// SIMATIC STEP 7 (V5.x) project Estacionamiento
// CPU: CPU 315-2 DP
// CPU: CPU 315-2 DP
// station: Hardware
// station: Estación 1
// station: P_ADR_BUS
// station: Hardware
// station: Estación 2
// station: P_ADR_BUS
// program: 2P
// program: Programa S7(6)
// program: Programa S7(7)

// (several symbol tables fit these blocks; global names not applied)

// FC 1: know-how protected block, not included

// FC 2: know-how protected block, not included

ORGANIZATION_BLOCK OB 1
TITLE = "Main Program Sweep (Cycle)"
VERSION : 0.1
VAR_TEMP
  OB1_EV_CLASS : BYTE ;	//Bits 0-3 = 1 (Coming event), Bits 4-7 = 1 (Event class 1)
  OB1_SCAN_1 : BYTE ;	//1 (Cold restart scan 1 of OB 1), 3 (Scan 2-n of OB 1)
  OB1_PRIORITY : BYTE ;	//Priority of OB Execution
  OB1_OB_NUMBR : BYTE ;	//1 (Organization block 1, OB1)
  OB1_RESERVED_1 : BYTE ;	//Reserved for system
  OB1_RESERVED_2 : BYTE ;	//Reserved for system
  OB1_PREV_CYCLE : INT ;	//Cycle time of previous OB1 scan (milliseconds)
  OB1_MIN_CYCLE : INT ;	//Minimum cycle time of OB1 (milliseconds)
  OB1_MAX_CYCLE : INT ;	//Maximum cycle time of OB1 (milliseconds)
  OB1_DATE_TIME : DATE_AND_TIME ;	//Date and time OB1 started
END_VAR
BEGIN
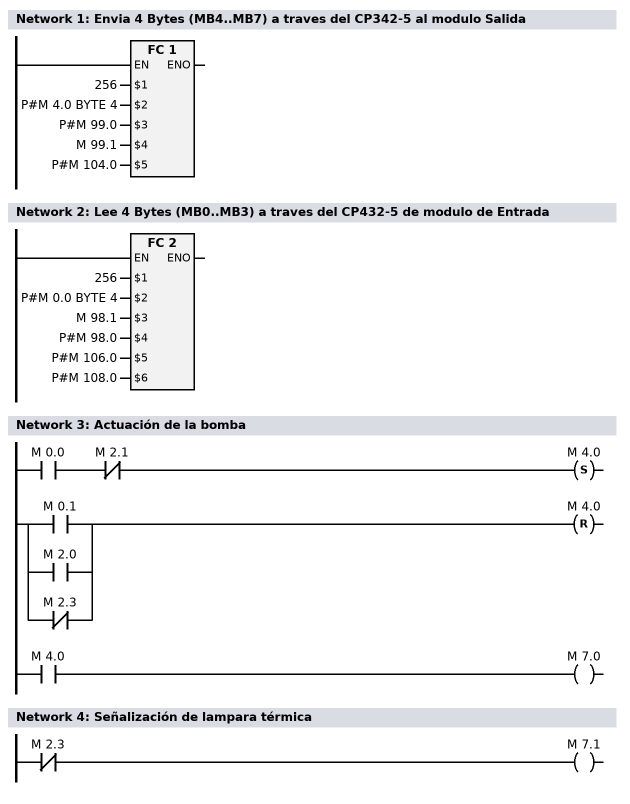
NETWORK
TITLE = Envia 4 Bytes (MB4..MB7) a traves del CP342-5 al modulo Salida
      CALL  FC 1 (
           $1                       := 256,
           $2                       := P#M 4.0 BYTE 4,
           $3                       := P#M 99.0,
           $4                       := M 99.1,
           $5                       := P#M 104.0);
      NOP   0;
NETWORK
TITLE = Lee 4 Bytes (MB0..MB3) a traves del CP432-5 de modulo de Entrada
      CALL  FC 2 (
           $1                       := 256,
           $2                       := P#M 0.0 BYTE 4,
           $3                       := M 98.1,
           $4                       := P#M 98.0,
           $5                       := P#M 106.0,
           $6                       := P#M 108.0);
      NOP   0;
NETWORK
TITLE = Actuación de la bomba
//Importante: Considerando el pulsador start tiene 
//autoretención. 
//Se inicia el sistema presionando el boton de start, 
//si el sensor bajo no detecta agua la bomba debe activarse.
//Si el sensor de alto detecta agua se debe apagar la bomba.
//Si se presiona el boton STOP la bomba debe parar.
//Si el sensor térmico esta activo tambien debe parar
//la bomba 
      A     M 0.0;
      AN    M 2.1;
      S     M 4.0;
      A(;
      O     M 0.1;
      O     M 2.0;
      ON    M 2.3;
      );
      R     M 4.0;
      A     M 4.0;
      =     M 7.0;
NETWORK
TITLE = Señalización de lampara térmica
//Si el sensor térmico esta activo se enciende la 
//señalización del Térmico
      AN    M 2.3;
      =     M 7.1;
NETWORK
TITLE =
END_ORGANIZATION_BLOCK

SYMBOL_TABLE
"Cuenta"	C 0	COUNTER	// Cantidad de vehículos estacionados
"DP_SEND"	FC 1	FC 1	// DP-SEND-Function for  SIMATIC NET CPs
"DP_RECV"	FC 2	FC 2	// DP-RECV-Function for  SIMATIC NET CPs
"ON/OFF Fisico"	I 0.0	BOOL	// Switch para modificar estado de la marca ON/OFF
"Reset Fisico"	I 0.1	BOOL	// Botón para resetear el contador
"Cont Entrada"	M 0.0	BOOL	// Aumenta el contador en uno al activarse (Corresponde con el I0.0)
"Cont Salida"	M 0.1	BOOL	// Disminuye el contador en uno al activarse (Corresponde con el I0.1)
"Lámpara Libre"	M 4.1	BOOL	// Se activa mientras estén menos de 20 vehículos dentro del estacionamiento (Q0.1)
"Lámpara Ocupado"	M 4.2	BOOL	// Se activa mientras estén 20 vehículos dentro del estacionamiento (Q0.2)
"Abrir"	M 5.0	BOOL	// Botón que libera el paso (Q1.0, en lugar del Q0.0 planteado inicialmente)
"Cerrar"	M 5.1	BOOL	// Botón que cierra el paso (Q1.1, en lugar del Q0.0 planteado inicialmente)
"ON/OFF"	M 30.0	BOOL	// Se activa el Sistema (ON) o cierra la barrera y conserva la cuenta (OFF) (input)
"Reset"	M 30.1	BOOL	// Vuelve a cero el contador (input físico o lógico)
"Marca Pizcando"	M 32.0	BOOL	// Para el pizcando de la luz
"Contador"	MW 102	WORD	// Cantidad de vehículos estacionados
"Cycle Execution"	OB 1	OB 1
"Hora"	QW 0	WORD
"Minuto"	QW 2	WORD
"READ_CLK"	SFC 1	SFC 1	// Read System Clock
"Temp"	T 0	TIMER	// Para la luz intermitente
"Temp1"	T 1	TIMER	// Para luz intermitente 2
END_SYMBOL_TABLE

// FC 1: know-how protected block, not included

// FC 2: know-how protected block, not included

ORGANIZATION_BLOCK "Cycle Execution"	// OB 1
TITLE = "Main Program Sweep (Cycle)"
VERSION : 0.1
VAR_TEMP
  OB1_EV_CLASS : BYTE ;	//Bits 0-3 = 1 (Coming event), Bits 4-7 = 1 (Event class 1)
  OB1_SCAN_1 : BYTE ;	//1 (Cold restart scan 1 of OB 1), 3 (Scan 2-n of OB 1)
  OB1_PRIORITY : BYTE ;	//Priority of OB Execution
  OB1_OB_NUMBR : BYTE ;	//1 (Organization block 1, OB1)
  OB1_RESERVED_1 : BYTE ;	//Reserved for system
  OB1_RESERVED_2 : BYTE ;	//Reserved for system
  OB1_PREV_CYCLE : INT ;	//Cycle time of previous OB1 scan (milliseconds)
  OB1_MIN_CYCLE : INT ;	//Minimum cycle time of OB1 (milliseconds)
  OB1_MAX_CYCLE : INT ;	//Maximum cycle time of OB1 (milliseconds)
  realtime : DATE_AND_TIME ;	//Date and time OB1 started
END_VAR
BEGIN
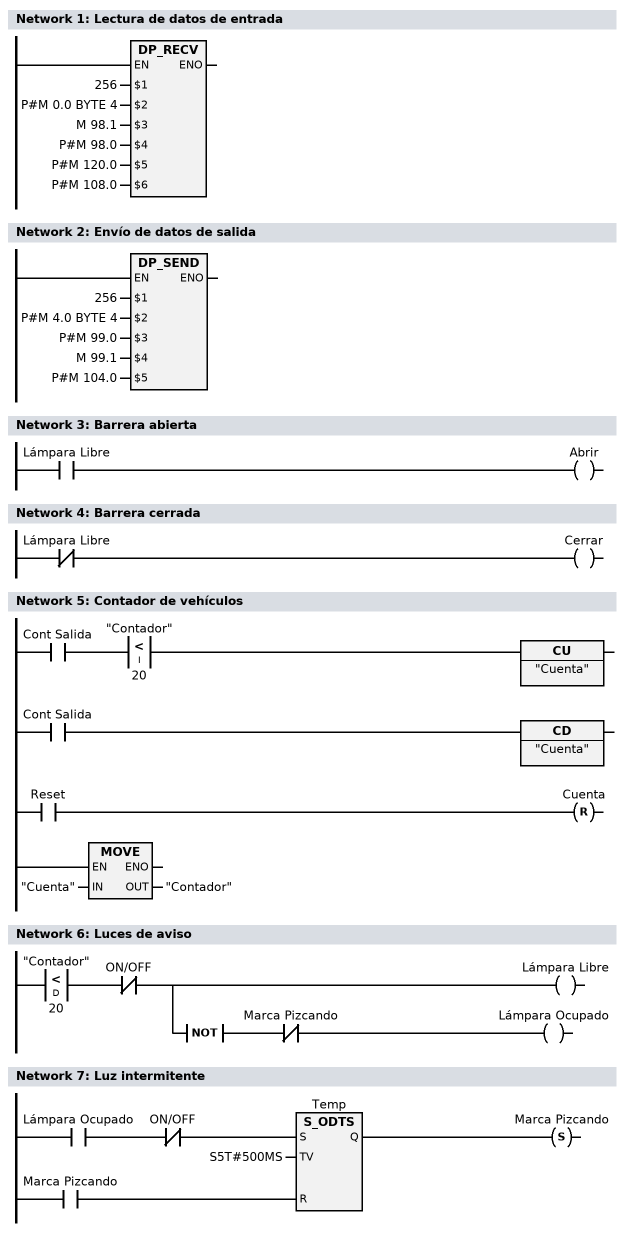
NETWORK
TITLE = Lectura de datos de entrada
      CALL  "DP_RECV" (
           $1                       := 256,
           $2                       := P#M 0.0 BYTE 4,
           $3                       := M 98.1,
           $4                       := P#M 98.0,
           $5                       := P#M 120.0,
           $6                       := P#M 108.0);
      NOP   0;
NETWORK
TITLE = Envío de datos de salida
      CALL  "DP_SEND" (
           $1                       := 256,
           $2                       := P#M 4.0 BYTE 4,
           $3                       := P#M 99.0,
           $4                       := M 99.1,
           $5                       := P#M 104.0);
      NOP   0;
NETWORK
TITLE = Barrera abierta
//Se mantine la barrera abierta mientras haya lugar ("lampara libre")
      A     "Lámpara Libre";
      =     "Abrir";
NETWORK
TITLE = Barrera cerrada
//Se mantine la barrera cerrada mientras no haya lugar ("lampara ocupada")
      AN    "Lámpara Libre";
      =     "Cerrar";
NETWORK
TITLE = Contador de vehículos
//Se realiza la deteccion de autos mediante los sensores del contador de 
//entrada/salida. El "cont entrada" aumente en 1 cuando ingresa un vehiculo;
//si el "Contador" es menor que la capacidad max. de autos (20)
//Y con el "cont salida" disminuye en 1 el "Contador" cuando sale un vehiculo.
      A     "Cont Salida";
      A(;
      L     "Contador";
      L     20;
      <I;
      );
      CU    "Cuenta";
      A     "Cont Salida";
      CD    "Cuenta";
      NOP   0;
      NOP   0;
      A     "Reset";
      R     "Cuenta";
      L     "Cuenta";
      T     "Contador";
      NOP   0;
      NOP   0;
NETWORK
TITLE = Luces de aviso
//Si el "Contador" es menor a 20 la "Lampara Libre" estara encendida
//y si llega a la capacidad maxima se enciende la "Lampara Ocupado" de 
//manera intermitente
      A(;
      L     "Contador";
      L     20;
      <D;
      );
      AN    "ON/OFF";
      =     L 20.0;
      A     L 20.0;
      BLD   102;
      =     "Lámpara Libre";
      A     L 20.0;
      NOT;
      AN    "Marca Pizcando";
      =     "Lámpara Ocupado";
NETWORK
TITLE = Luz intermitente
//Metodo por el cual se logra que la "Lampara Ocupado"
//se encienda de forma intermitente parte 1
      A     "Lámpara Ocupado";
      AN    "ON/OFF";
      L     S5T#500MS;
      SS    "Temp";
      A     "Marca Pizcando";
      R     "Temp";
      NOP   0;
      NOP   0;
      A     "Temp";
      S     "Marca Pizcando";
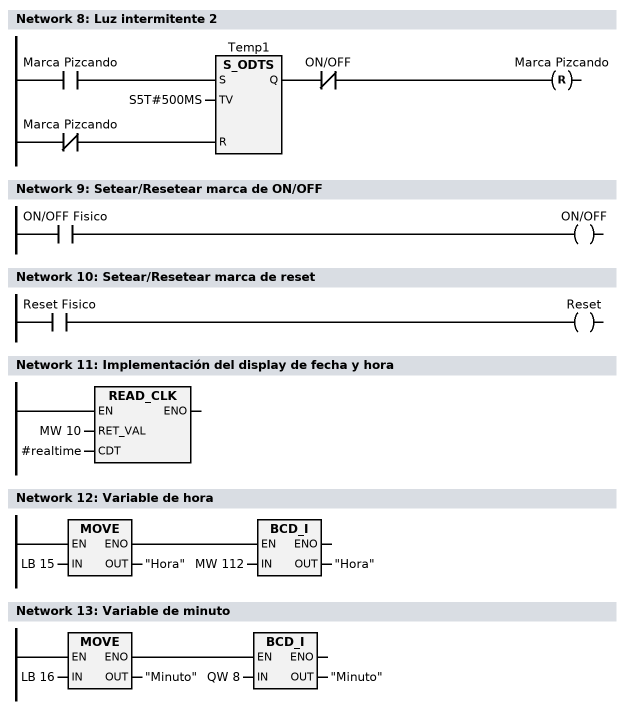
NETWORK
TITLE = Luz intermitente 2
//Metodo por el cual se logra que la "Lampara Ocupado"
//se encienda de forma intermitente parte 2
      A(;
      A     "Marca Pizcando";
      L     S5T#500MS;
      SS    "Temp1";
      AN    "Marca Pizcando";
      R     "Temp1";
      NOP   0;
      NOP   0;
      A     "Temp1";
      );
      AN    "ON/OFF";
      R     "Marca Pizcando";
NETWORK
TITLE = Setear/Resetear marca de ON/OFF
//Una vez que se cambia el valor del switch físico de on/off, una marca toma ese 
//valor. Este switch se encuentra del lado de la CPU.
      A     "ON/OFF Fisico";
      =     "ON/OFF";
NETWORK
TITLE = Setear/Resetear marca de reset
//Así como el switch de on/off, el botón físico de reset se encuentra del lado 
//del 
//operador (donde está el CPU), y la marca se activa mientras el botón esté 
//pulsado.
      A     "Reset Fisico";
      =     "Reset";
NETWORK
TITLE = Implementación del display de fecha y hora
//Los siguientes segmentos asignarán valores codificados en BCD del  
//hora y minuto para que estos sean mostrados del lado del 
//CPU, conectando estas salidas físicas a displays de 7 segmentos que reciban 
//números en BCD como entradas.
      CALL  "READ_CLK" (
           RET_VAL                  := MW 10,
           CDT                      := #realtime);
      NOP   0;
NETWORK
TITLE = Variable de hora
      A(;
      L     LB 15;
      T     "Hora";
      SET;
      SAVE;
      CLR;
      A     BR;
      );
      JNB   _001;
      L     MW 112;
      BTI;
      T     "Hora";
_001: NOP   0;
NETWORK
TITLE = Variable de minuto
      A(;
      L     LB 16;
      T     "Minuto";
      SET;
      SAVE;
      CLR;
      A     BR;
      );
      JNB   _002;
      L     QW 8;
      BTI;
      T     "Minuto";
_002: NOP   0;
END_ORGANIZATION_BLOCK

SYMBOL_TABLE
"DP_SEND"	FC 1	FC 1	// DP-SEND-Function for  SIMATIC NET CPs
"DP_RECV"	FC 2	FC 2	// DP-RECV-Function for  SIMATIC NET CPs
"AG_SEND"	FC 5	FC 5	// AG SEND
"AG_RECV"	FC 6	FC 6	// AG RECEIVE
"Cycle Execution"	OB 1	OB 1
"READ_CLK"	SFC 1	SFC 1	// Read System Clock
END_SYMBOL_TABLE

// FC 5: know-how protected block, not included

// FC 6: know-how protected block, not included

ORGANIZATION_BLOCK "Cycle Execution"	// OB 1
TITLE = "Main Program Sweep (Cycle)"
VERSION : 0.1
VAR_TEMP
  OB1_EV_CLASS : BYTE ;	//Bits 0-3 = 1 (Coming event), Bits 4-7 = 1 (Event class 1)
  OB1_SCAN_1 : BYTE ;	//1 (Cold restart scan 1 of OB 1), 3 (Scan 2-n of OB 1)
  OB1_PRIORITY : BYTE ;	//Priority of OB Execution
  OB1_OB_NUMBR : BYTE ;	//1 (Organization block 1, OB1)
  OB1_RESERVED_1 : BYTE ;	//Reserved for system
  OB1_RESERVED_2 : BYTE ;	//Reserved for system
  OB1_PREV_CYCLE : INT ;	//Cycle time of previous OB1 scan (milliseconds)
  OB1_MIN_CYCLE : INT ;	//Minimum cycle time of OB1 (milliseconds)
  OB1_MAX_CYCLE : INT ;	//Maximum cycle time of OB1 (milliseconds)
  realtime : DATE_AND_TIME ;	//Date and time OB1 started
END_VAR
BEGIN
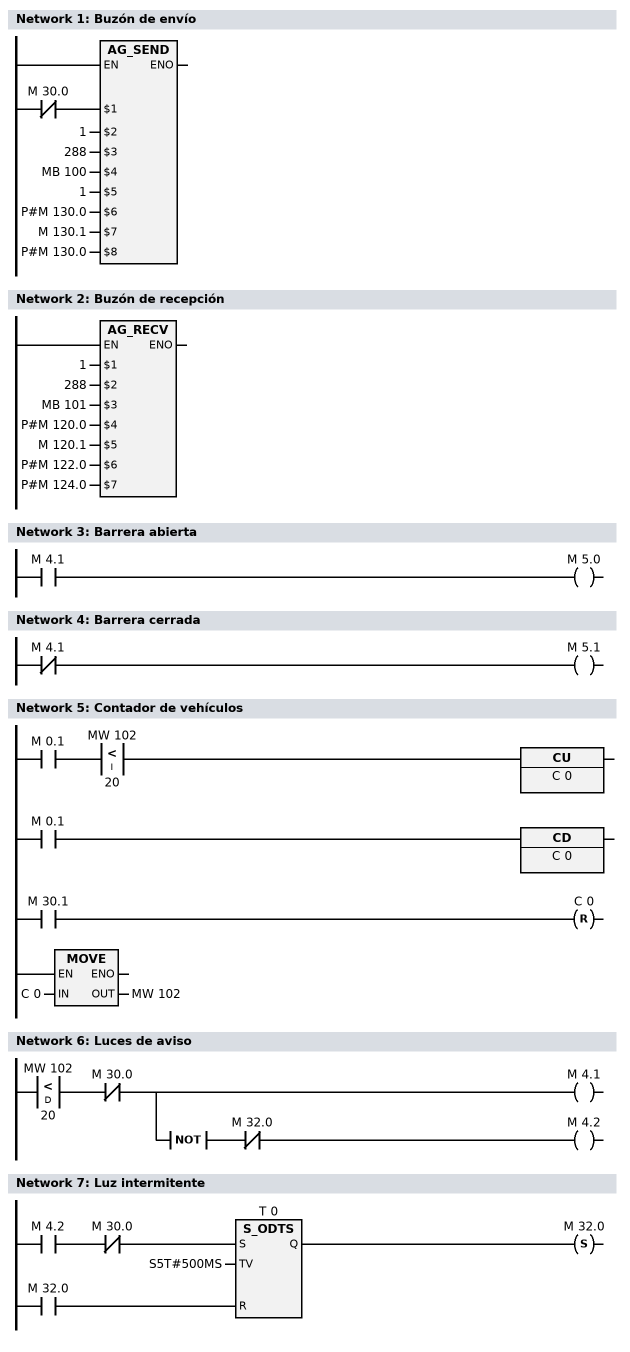
NETWORK
TITLE = Buzón de envío
      AN    M 30.0;
      =     L 20.0;
      BLD   103;
      CALL  "AG_SEND" (
           $1                       := L 20.0,
           $2                       := 1,
           $3                       := 288,
           $4                       := MB 100,
           $5                       := 1,
           $6                       := P#M 130.0,
           $7                       := M 130.1,
           $8                       := P#M 130.0);
      NOP   0;
NETWORK
TITLE = Buzón de recepción
      CALL  "AG_RECV" (
           $1                       := 1,
           $2                       := 288,
           $3                       := MB 101,
           $4                       := P#M 120.0,
           $5                       := M 120.1,
           $6                       := P#M 122.0,
           $7                       := P#M 124.0);
      NOP   0;
NETWORK
TITLE = Barrera abierta
//Se mantine la barrera abierta mientras haya lugar ("lampara libre")
      A     M 4.1;
      =     M 5.0;
NETWORK
TITLE = Barrera cerrada
//Se mantine la barrera cerrada mientras no haya lugar ("lampara ocupada")
      AN    M 4.1;
      =     M 5.1;
NETWORK
TITLE = Contador de vehículos
//Se realiza la deteccion de autos mediante los sensores del contador de 
//entrada/salida. El "cont entrada" aumente en 1 cuando ingresa un vehiculo;
//si el "Contador" es menor que la capacidad max. de autos (20)
//Y con el "cont salida" disminuye en 1 el "Contador" cuando sale un vehiculo.
      A     M 0.1;
      A(;
      L     MW 102;
      L     20;
      <I;
      );
      CU    C 0;
      A     M 0.1;
      CD    C 0;
      NOP   0;
      NOP   0;
      A     M 30.1;
      R     C 0;
      L     C 0;
      T     MW 102;
      NOP   0;
      NOP   0;
NETWORK
TITLE = Luces de aviso
//Si el "Contador" es menor a 20 la "Lampara Libre" estara encendida
//y si llega a la capacidad maxima se enciende la "Lampara Ocupado" de 
//manera intermitente
      A(;
      L     MW 102;
      L     20;
      <D;
      );
      AN    M 30.0;
      =     L 20.0;
      A     L 20.0;
      BLD   102;
      =     M 4.1;
      A     L 20.0;
      NOT;
      AN    M 32.0;
      =     M 4.2;
NETWORK
TITLE = Luz intermitente
//Metodo por el cual se logra que la "Lampara Ocupado"
//se encienda de forma intermitente parte 1
      A     M 4.2;
      AN    M 30.0;
      L     S5T#500MS;
      SS    T 0;
      A     M 32.0;
      R     T 0;
      NOP   0;
      NOP   0;
      A     T 0;
      S     M 32.0;
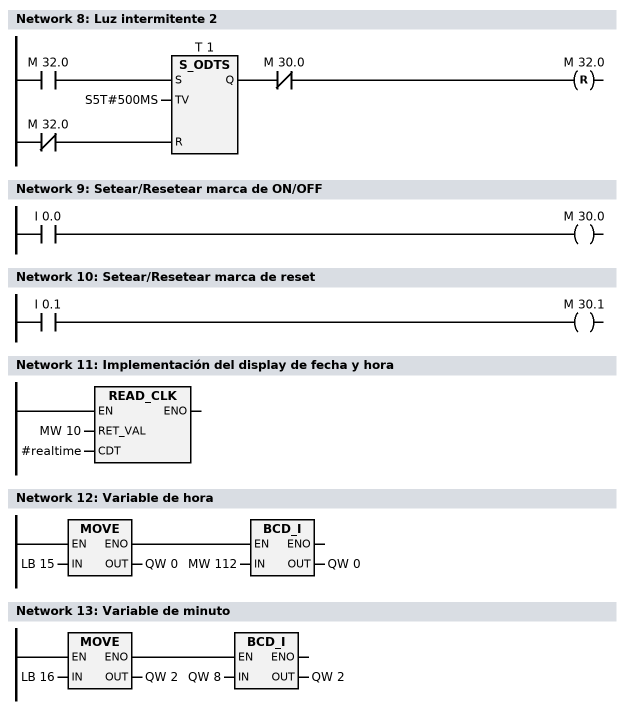
NETWORK
TITLE = Luz intermitente 2
//Metodo por el cual se logra que la "Lampara Ocupado"
//se encienda de forma intermitente parte 2
      A(;
      A     M 32.0;
      L     S5T#500MS;
      SS    T 1;
      AN    M 32.0;
      R     T 1;
      NOP   0;
      NOP   0;
      A     T 1;
      );
      AN    M 30.0;
      R     M 32.0;
NETWORK
TITLE = Setear/Resetear marca de ON/OFF
//Una vez que se cambia el valor del switch físico de on/off, una marca toma ese 
//valor. Este switch se encuentra del lado de la CPU.
      A     I 0.0;
      =     M 30.0;
NETWORK
TITLE = Setear/Resetear marca de reset
//Así como el switch de on/off, el botón físico de reset se encuentra del lado 
//del 
//operador (donde está el CPU), y la marca se activa mientras el botón esté 
//pulsado.
      A     I 0.1;
      =     M 30.1;
NETWORK
TITLE = Implementación del display de fecha y hora
//Los siguientes segmentos asignarán valores codificados en BCD del  
//hora y minuto para que estos sean mostrados del lado del 
//CPU, conectando estas salidas físicas a displays de 7 segmentos que reciban 
//números en BCD como entradas.
      CALL  "READ_CLK" (
           RET_VAL                  := MW 10,
           CDT                      := #realtime);
      NOP   0;
NETWORK
TITLE = Variable de hora
      A(;
      L     LB 15;
      T     QW 0;
      SET;
      SAVE;
      CLR;
      A     BR;
      );
      JNB   _001;
      L     MW 112;
      BTI;
      T     QW 0;
_001: NOP   0;
NETWORK
TITLE = Variable de minuto
      A(;
      L     LB 16;
      T     QW 2;
      SET;
      SAVE;
      CLR;
      A     BR;
      );
      JNB   _002;
      L     QW 8;
      BTI;
      T     QW 2;
_002: NOP   0;
END_ORGANIZATION_BLOCK

SYMBOL_TABLE
"AG_SEND"	FC 5	FC 5	// AG SEND
"AG_RECV"	FC 6	FC 6	// AG RECEIVE
END_SYMBOL_TABLE

// FC 5: know-how protected block, not included

// FC 6: know-how protected block, not included

ORGANIZATION_BLOCK OB 1
TITLE = "Main Program Sweep (Cycle)"
VERSION : 0.1
VAR_TEMP
  OB1_EV_CLASS : BYTE ;	//Bits 0-3 = 1 (Coming event), Bits 4-7 = 1 (Event class 1)
  OB1_SCAN_1 : BYTE ;	//1 (Cold restart scan 1 of OB 1), 3 (Scan 2-n of OB 1)
  OB1_PRIORITY : BYTE ;	//Priority of OB Execution
  OB1_OB_NUMBR : BYTE ;	//1 (Organization block 1, OB1)
  OB1_RESERVED_1 : BYTE ;	//Reserved for system
  OB1_RESERVED_2 : BYTE ;	//Reserved for system
  OB1_PREV_CYCLE : INT ;	//Cycle time of previous OB1 scan (milliseconds)
  OB1_MIN_CYCLE : INT ;	//Minimum cycle time of OB1 (milliseconds)
  OB1_MAX_CYCLE : INT ;	//Maximum cycle time of OB1 (milliseconds)
  OB1_DATE_TIME : DATE_AND_TIME ;	//Date and time OB1 started
END_VAR
BEGIN
NETWORK
TITLE = Buzón de envío
      AN    M 30.0;
      =     L 20.0;
      BLD   103;
      CALL  "AG_SEND" (
           $1                       := L 20.0,
           $2                       := 1,
           $3                       := 288,
           $4                       := MB 103,
           $5                       := 1,
           $6                       := P#M 130.0,
           $7                       := M 130.1,
           $8                       := P#M 130.0);
      NOP   0;
NETWORK
TITLE = Buzón de recepción
      CALL  "AG_RECV" (
           $1                       := 1,
           $2                       := 288,
           $3                       := MB 102,
           $4                       := P#M 120.0,
           $5                       := M 120.1,
           $6                       := P#M 122.0,
           $7                       := P#M 124.0);
      NOP   0;
END_ORGANIZATION_BLOCK
